Fanuc TP program (LS listing): UP206.LS

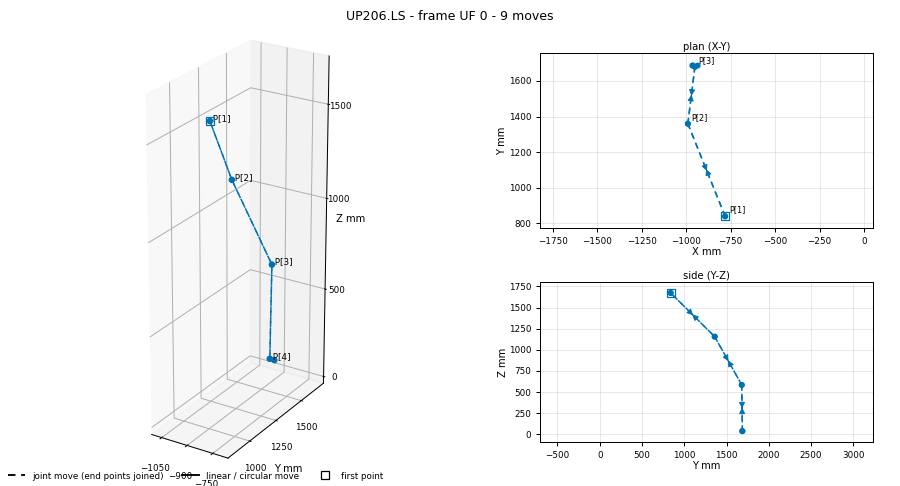
[picture p0: tool path of UP206.LS in frame UF 0, 9 of 9 moves have a stored position in this frame; points joined in program order, loops and branches not executed]
/PROG  UP206
/ATTR
OWNER		= AUROM;
COMMENT		= "Prueba TCP SP1";
PROG_SIZE	= 3526;
CREATE		= DATE 96-03-15  TIME 09:24:00;
MODIFIED	= DATE 17-05-23  TIME 06:23:14;
FILE_NAME	= UP101;
VERSION		= 0;
LINE_COUNT	= 16;
MEMORY_SIZE	= 7134;
PROTECT		= READ_WRITE;
TCD:  STACK_SIZE	= 500,
      TASK_PRIORITY	= 50,
      TIME_SLICE	= 0,
      BUSY_LAMP_OFF	= 0,
      ABORT_REQUEST	= 0,
      PAUSE_REQUEST	= 0;
DEFAULT_GROUP	= 1,1,1,1,*;
CONTROL_CODE	= 00000000 00000000;
/APPL
/MN
   1:  UTOOL_NUM=24 ;
   2:  UFRAME_NUM=0 ;
   3:  PAYLOAD[1] ;
   4:J P[1] 100% CNT0 ACC100 TB    .10sec,P-SPS    ;
      1:  TC_ONLINE (ON) ;
      2:  DO[23]=OFF ;
      3:  CALL MAKRO050    ;
      4:  WAIT (DO[11])    ;
      5:  WAIT (DI[23])    ;
      6:  DO[23]=ON ;
      7:  TC_ONLINE (DO[11] AND M[30] AND M[95]) ;
       ------ ;
   5:J P[2] 100% CNT100 ACC100 TB   0.00sec,P-SPS    ;
      1:  TC_ONLINE (DO[11] AND M[30] AND M[95]) ;
       ------ ;
   6:J P[3] 100% CNT100 ACC100 TB   0.00sec,P-SPS    ;
      1:  TC_ONLINE (DO[11] AND M[30] AND M[95]) ;
       ------ ;
   7:J P[4] 100% CNT0 ACC100 TB    .10sec,P-SPS    ;
      1:  TC_ONLINE (ON) ;
      2:  DO[23]=OFF ;
      3:  WAIT (DI[23])    ;
      4:  DO[23]=ON ;
      5:  TC_ONLINE (DO[11] AND M[30] AND M[95]) ;
       ------ ;
   8:  !Posicion Prueba TCP ;
   9:  !SP1 ;
  10:  !X=-934.119 Y=1702.416 Z=-1073.87 ;
  11:  !W=-179.266 P=1.389 R=.248 ;
  12:L P[5] 400mm/sec CNT0 ACC100 TB    .10sec,P-SPS    ;
      1:  TC_ONLINE (ON) ;
      2:  DO[23]=OFF ;
      3:  WAIT (DI[17])    ;
      4:  WAIT (DI[23])    ;
      5:  DO[23]=ON ;
      6:  TC_ONLINE (DO[11] AND M[30] AND M[95]) ;
       ------ ;
  13:L P[6] 400mm/sec CNT0 ACC100 TB    .10sec,P-SPS    ;
      1:  TC_ONLINE (ON) ;
      2:  DO[23]=OFF ;
      3:  WAIT (DI[23])    ;
      4:  DO[23]=ON ;
      5:  TC_ONLINE (DO[11] AND M[30] AND M[95]) ;
       ------ ;
  14:J P[7] 100% CNT100 ACC100 TB   0.00sec,P-SPS    ;
      1:  TC_ONLINE (DO[11] AND M[30] AND M[95]) ;
       ------ ;
  15:J P[8] 100% CNT100 ACC100 TB   0.00sec,P-SPS    ;
      1:  TC_ONLINE (DO[11] AND M[30] AND M[95]) ;
       ------ ;
  16:J P[9] 100% CNT0 ACC100 TB    .10sec,P-SPS    ;
      1:  TC_ONLINE (ON) ;
      2:  DO[23]=OFF ;
      3:  WAIT (DI[23])    ;
      4:  DO[23]=ON ;
      5:  TC_ONLINE (DO[11] AND M[30] AND M[95]) ;
       ------ ;
/POS
P[1]{
   GP1:
	UF : 0, UT : 24,		CONFIG : 'N U T, 0, 0, 0',
	X =  -781.134  mm,	Y =   838.843  mm,	Z =  1672.802  mm,
	W =   172.006 deg,	P =    30.544 deg,	R =   -79.872 deg
   GP2:
	UF : 0, UT : 1,
	J1=   100.000  mm
   GP3:
	UF : 0, UT : 1,
	J1=     0.000  mm
   GP4:
	UF : 0, UT : 1,
	J1=     0.000  mm
};
P[2]{
   GP1:
	UF : 0, UT : 24,		CONFIG : 'N U T, 0, 0, 1',
	X =  -990.840  mm,	Y =  1359.610  mm,	Z =  1155.815  mm,
	W =  -171.178 deg,	P =    12.442 deg,	R =   -33.320 deg
   GP2:
	UF : 0, UT : 1,
	J1=   100.000  mm
   GP3:
	UF : 0, UT : 1,
	J1=     0.000  mm
   GP4:
	UF : 0, UT : 1,
	J1=     0.000  mm
};
P[3]{
   GP1:
	UF : 0, UT : 24,		CONFIG : 'N U T, 0, 0, 1',
	X =  -951.052  mm,	Y =  1679.725  mm,	Z =   584.914  mm,
	W =  -179.266 deg,	P =     1.388 deg,	R =      .248 deg
   GP2:
	UF : 0, UT : 1,
	J1=   100.000  mm
   GP3:
	UF : 0, UT : 1,
	J1=     0.000  mm
   GP4:
	UF : 0, UT : 1,
	J1=     0.000  mm
};
P[4]{
   GP1:
	UF : 0, UT : 24,		CONFIG : 'N U T, 0, 0, 1',
	X =  -964.324  mm,	Y =  1686.667  mm,	Z =    38.537  mm,
	W =  -179.266 deg,	P =     1.388 deg,	R =      .248 deg
   GP2:
	UF : 0, UT : 1,
	J1=   100.000  mm
   GP3:
	UF : 0, UT : 1,
	J1=     0.000  mm
   GP4:
	UF : 0, UT : 1,
	J1=     0.000  mm
};
P[5]{
   GP1:
	UF : 0, UT : 24,		CONFIG : 'N U T, 0, 0, 1',
	X =  -935.704  mm,	Y =  1686.424  mm,	Z =    37.503  mm,
	W =  -179.266 deg,	P =     1.388 deg,	R =      .248 deg
   GP2:
	UF : 0, UT : 1,
	J1=   100.000  mm
   GP3:
	UF : 0, UT : 1,
	J1=     0.000  mm
   GP4:
	UF : 0, UT : 1,
	J1=     0.000  mm
};
P[6]{
   GP1:
	UF : 0, UT : 24,		CONFIG : 'N U T, 0, 0, 1',
	X =  -964.324  mm,	Y =  1686.667  mm,	Z =    38.537  mm,
	W =  -179.266 deg,	P =     1.388 deg,	R =      .248 deg
   GP2:
	UF : 0, UT : 1,
	J1=   100.000  mm
   GP3:
	UF : 0, UT : 1,
	J1=     0.000  mm
   GP4:
	UF : 0, UT : 1,
	J1=     0.000  mm
};
P[7]{
   GP1:
	UF : 0, UT : 24,		CONFIG : 'N U T, 0, 0, 1',
	X =  -951.052  mm,	Y =  1679.725  mm,	Z =   584.914  mm,
	W =  -179.266 deg,	P =     1.388 deg,	R =      .248 deg
   GP2:
	UF : 0, UT : 1,
	J1=   100.000  mm
   GP3:
	UF : 0, UT : 1,
	J1=     0.000  mm
   GP4:
	UF : 0, UT : 1,
	J1=     0.000  mm
};
P[8]{
   GP1:
	UF : 0, UT : 24,		CONFIG : 'N U T, 0, 0, 1',
	X =  -990.840  mm,	Y =  1359.610  mm,	Z =  1155.815  mm,
	W =  -171.178 deg,	P =    12.442 deg,	R =   -33.320 deg
   GP2:
	UF : 0, UT : 1,
	J1=   100.000  mm
   GP3:
	UF : 0, UT : 1,
	J1=     0.000  mm
   GP4:
	UF : 0, UT : 1,
	J1=     0.000  mm
};
P[9]{
   GP1:
	UF : 0, UT : 24,		CONFIG : 'N U T, 0, 0, 0',
	X =  -781.134  mm,	Y =   838.843  mm,	Z =  1672.802  mm,
	W =   172.006 deg,	P =    30.544 deg,	R =   -79.872 deg
   GP2:
	UF : 0, UT : 1,
	J1=   100.000  mm
   GP3:
	UF : 0, UT : 1,
	J1=     0.000  mm
   GP4:
	UF : 0, UT : 1,
	J1=     0.000  mm
};
/END
